// TIA Portal V17 export
// export: Created 2023-12-22T15:04:45.1849706Z, ExportSetting WithDefaults, DisplayName Totally Integrated Automation Portal, DisplayVersion V17, DisplayName TIA Portal Openness, DisplayVersion V17, DisplayName TIA Portal Version Control Interface, DisplayVersion V17, DisplayName STEP 7 Professional, DisplayVersion V17, DisplayName STEP 7 Safety, DisplayVersion V17, DisplayName WinCC Advanced, DisplayVersion V17
DATA_BLOCK "System_DB"   // DB4
VERSION : 0.1
// stored: AutoNumber true, DBAccessibleFromOPCUA true, InstanceOfName System, InstanceOfType FB
"System"
   // VAR
   //    PE_1_Delta : Real;
   //    PE_2_Detla : Real;
   //    PE_1_Min : Real;
   //    PE_2_Min : Real;
   // END_VAR
BEGIN
END_DATA_BLOCK
